FUNCTION_BLOCK InputAts400 IMPLEMENTS IInputAts400
VAR_INPUT
    input : ARRAY[1..8] OF BOOL;
END_VAR

METHOD GetInputData : InputDataAts400
VAR_INPUT
END_VAR
GetInputData.Pass          := input[1];
GetInputData.Fail          := input[2];
GetInputData.InOp          := input[3];
GetInputData.ResultImpuls  := input[4];
GetInputData.DummyOut      := input[5];
GetInputData.Ready         := input[6];
GetInputData.SafetyCircuit := input[7];
GetInputData.ContactExits  := input[8];
END_METHOD

END_FUNCTION_BLOCK

(* stored: Version 1.1.0.1, ProductVersion 3.1.4024.12
   POU InputAts400: Id {5d570cb8-20ee-4157-98b1-95e06e64bd2c}, SpecialFunc None
   Method GetInputData: Id {b0529c67-6ace-40e9-ac29-5bc133d8a1d9} *)
